PROGRAM PRG_Main
VAR
	bTestInput: BOOL;
	bTestOutput: BOOL;
	fbMachine: FB_ExampleMachine;
	fbStation1: FB_ExampleStation;
	fbStation2: FB_ExampleStation;
	fbStation3: FB_ExampleStation;
	fbStation4: FB_ExampleStation;
	bStart: BOOL;
	bAbort: BOOL;
	bReset: BOOL;
	bStop: BOOL;
	bSuspend: BOOL;
	fbDevice1: FB_ExampleDevice;
	fbDevice2: FB_ExampleDevice;
	fbDevice3: FB_ExampleDevice;
	fbDevice4: FB_ExampleDevice;
	bPoweredOn: BOOL;
//	FB_AdsDeviceAPI_0: FB_AdsDeviceAPI;
	FB_AdsDeviceAPI_0 : FB_AdsCommandRouter;
//	FB_AdsDeviceAPI_1 : FB_AdsCommandRouter;
	MyLaser1: FB_KeyenceLaserMarkerMDX2000;
	(* Database handler FB. *)
//	in_fbDataHandler: REFERENCE TO FB_Data;
	bConnectToLaserMarker: BOOL;
	bRes_LaserConnected: BOOL;
	bTestADSServer: BOOL;
	strTarget: T_MaxString;
	strCommand: T_MaxString;
	arrParams: T_ApiMethodParameters;
	MyResults: T_MaxString;
	bInterfaceTest : BOOL;
	temp: BOOL;
	bDisconnectFromLaserMarker: BOOL;
	bRes_LaserDisconnected: BOOL;
	bPeakCurrentProgramInLaser: BOOL;
	bRes_PeakCurrentProgramInLaser: BOOL;
	bSendProgramToLaser: BOOL;
	bRes_SendProgramtoLaser: BOOL;
	filepath : STRING;
	LaserMemoryLocation : INT;
	bSaveCurrentLaserProgramtoPC : BOOL;
	bRes_SaveCurrentLaserProgramtoPC: BOOL;
	LaserProgramFolderPath: STRING;
	bGetCurrentProgram : BOOL;
	bRes_GetCurrentProgram : BOOL;
	CurrentProgramName : T_MaxString;
	bStartMarking: BOOL;
	bRes_StartMarking: BOOL;
	bStopMarking: BOOL;
	bRes_StopMarking: BOOL;
	bClearLaserErrors: BOOL;
	bRes_ClearLaserErrors: BOOL;
	bUpdateProgramBlockInTheLaser: BOOL;
	bRes_UpdateProgramBlockInTheLaser: BOOL;
	_blockNumber: INT;
	_blockData: STRING;
	_blockType : BlockTypes;
	bGetLaserStatus: BOOL;
	bRes_GetLaserStatus: BOOL;
	_string_laserstatus : STRING;
	bGetLaserErrorStatus: BOOL;
	bRes_GetLaserErrorStatus: BOOL;
	_bIsLaserError : BOOL;
	bGetLaserActivatedStatus: BOOL;
	bRes_GetLaserActivatedStatus: BOOL;
	_bIsLaserActivated : BOOL;
	bGetLaserMarkingStatus: BOOL;
	bRes_GetLaserMarkingStatus: BOOL;
	_bIsLaserMarking : BOOL;
	bRes_Reset: BOOL;
	bResetErrors: BOOL;
	bUpdateProgramBlockMarkEnabledInTheLaser: BOOL;
	bRes_UpdateProgramBlockMarkEnabledInTheLaser: BOOL;
	_bool_markenabled : BOOL;
	_blockType_enum : BlockTypes;
	UpdateSingleBlockMarkEnabledIntheLaser_Success: BOOL;
	_bUpdateSingleBlockDataSuccess : BOOL;
	_bUpdateSingleBlockMarkEnabled_Success : BOOL;
	bUpdateAllMarkingInfo: BOOL;
	LastBlockToMark : INT;
	_OneTimeArrayBuild : BOOL := TRUE;
	BlockInfoArray : ARRAY [0..255] OF OneBlockInfo;
	bRes_UpdateAllMarkingInfo: BOOL;
	intIndex: INT;
	intIndex2 : INT;
	inst_intStep: INT := 0;
	_tempString : STRING;
	bRes_UpdateAllMarkInfo : ARRAY [0..255] OF BOOL;
	bUpdateAllMarkingInfo_MethodCall: BOOL;
	bRes_UpdateAllMarkingInfo_MethodCall: BOOL;
	fbDataHandler: FB_DataTracker;
	fbDataHandler2: FB_DataTracker;
	fbDatabaseCommandRouter: FB_AdsCommandRouter;
	_inst_bDataTransferred: BOOL;
	// (* Name of the parameters database transfer ID. *)
	in_strParametersDatabaseName: T_MaxString := 'GetLimits';
	in_strParametersDBNameLaserLimits_L1 : T_MaxString := 'GetLaserMarkingParams_L1';
	in_strParametersDBNameLaserLimits_L2 : T_MaxString := 'GetLaserMarkingParams_L2';
	in_strParametersDBNameLaserLimits_R1 : T_MaxString := 'GetLaserMarkingParams_R1';
	in_strParametersDBNameLaserLimits_R2 : T_MaxString := 'GetLaserMarkingParams_R2';	
	_inst_bLaserLimitsDataTransferred_L1 : BOOL;
	_inst_bLaserLimitsDataTransferred_L2 : BOOL;
	_inst_bLaserLimitsDataTransferred_R1 : BOOL;
	_inst_bLaserLimitsDataTransferred_R2 : BOOL;
	bGetLimitsFromDB : BOOL;
	bGetLaserParamsFromDB_L1 : BOOL;
	bGetLaserParamsFromDB_L2 : BOOL;
	bGetLaserParamsFromDB_R1 : BOOL;
	bGetLaserParamsFromDB_R2 : BOOL;
	bPerformPriorOp_Smart: BOOL;
	in_strParametersDBName_SmartWater : T_MaxString := 'GetPriorOPA';
	_inst_bPriorOp_Smart: BOOL;
	
	bPerformPriorOp_FFT: BOOL;
	in_strParametersDBName_FFTLaser_L1 : T_MaxString := 'LaserMarkCheckL1';
	_inst_bPriorOp_FFT: BOOL;
	
	Temp_CR_LOOKUP_NestL1 : INT;
	iLengthDataMatrixNestL1 : INT;
	ParamsArrayNestA : STRING;
	
	//MES Data Tracking Testing
//	fbDataHandler3: FB_MESDataTracking;
	bPerformGetLotInfoFromLotBarcode: BOOL;
	_inst_bGetLotInfo_LotBarcode: BOOL;
	in_strParamDBName_GetLotInfo: T_MaxString := 'GetLotInfo1';
	
	bPerformGetOpInfoFromOpBarcode: BOOL;
	in_strParamDBName_GetOpInfo: T_MaxString := 'GetOperatorInfo1';
	_inst_bGetOpInfo_OpBarcode: BOOL;
	
	bPerformStartLot : BOOL;
	_inst_bStartLot : BOOL;
	in_strParamDBName_StartLot : T_MaxString := 'StartLot1';
	
	bPerformGetProdLotComponents : BOOL;
	_inst_bGetProdLotComponents : BOOL;
	in_strParamDBName_GetProdLotComps : T_MaxString := 'GetProdLotComponents1';
	
	bPerformComponentValidation1 : BOOL;
	_inst_bCompValidation1 : BOOL;
	in_strParamDBName_Comp1Validation1 : T_MaxString := 'ComponentValidation1';
	
	bPerformComponentValidation2 : BOOL;
	_inst_bCompValidation2 : BOOL;
	in_strParamDBName_Comp1Validation2 : T_MaxString := 'ComponentValidation2';
	
	bPerformComponentValidation3 : BOOL;
	_inst_bCompValidation3 : BOOL;
	in_strParamDBName_Comp1Validation3 : T_MaxString := 'ComponentValidation3';
	
	bPerformGetMachineSettings : BOOL;
	_inst_bGetMachineSettings : BOOL;
	in_strParamDBName_GetMachSetting : T_MaxString := 'GetMachineSettings1';
	
	bPerformAddScrapCompByReason : BOOL;
	_inst_bAddScrapCompByReason : BOOL;
	in_strParamDBName_AddScrapCompByReason : T_MaxString := 'AddScrapComponentByReason1';
	
	bPerformEndLotComp : BOOL;
	_inst_bEndLotComp : BOOL;
	in_strParamDBName_EndLotComp : T_MaxString := 'EndLotComponent1';
	
	bPerformGetMachineDefects : BOOL;
	_inst_bGetMachineDefects : BOOL;
	in_strParamDBName_GetMachDefects : T_MaxString := 'GetMachineDefects1';

	//Testing Cohap Related Vars

	//Initialize Only	
	MyCohapTest : FB_COHAP;
	bInitializeCohapSystem: BOOL;
	bRes_CohapConnected: BOOL;

	//Execute RunImpMethods Only	;
	bExecuteRunImpMethods: BOOL;
	bRes_RunImpMethods: BOOL;

	//Set Current Device Instance
	bSetCurrentDevice_Cohap : BOOL;
	bRes_SetCurrentDevice : BOOL;
	//Input Params
	strDeviceName : STRING;
	
	//RunCommand
	bRunCommandCohapSystem : BOOL;
	bRes_RunCommand : BOOL;
	//Input Params
	strMethodName : STRING;
	RunCom_InpuParams : T_CohapParameterList;
	RunCom_ExpOutParamList : ARRAY[0..2] OF ReturnParamKVP;
	//Output Params
	RunCom_OutputParams : T_CohapParameterList;
	
	//DummyTest Dictionary Prep for RunCommand Execution
	RC_DT_InpPar : T_CohapParameterList;
	RC_DT_ExpOutPL : ARRAY[0..2] OF ReturnParamKVP;
	
	CohapMethodStrings : TMethodNames_Cohap;
	CohapMethodControls : TMethod_Controls;
//	fbCohapHandler1: FB_COHAP;

///////////////////////////////

	// For readSerialNumber
	readSerialNumber_inpuparams : T_CohapParameterList;// := [(strKey: 'channel', strValue: '1'), (), ()];
	readSerialNumber_expoutparamlist : ARRAY[0..2] OF ReturnParamKVP;// := [(VarName: 'serialnumber', DataType: DT_UINT), (), ()];
	readSerialNumber_outputparams : T_CohapParameterList;// := [(), (), ()];
	
	// For ReadDeviceOutput
	ReadDeviceOutput_inpuparams : T_CohapParameterList;// := [(strKey: 'Channel', strValue: '10'), (), ()];
	ReadDeviceOutput_expoutparamlist : ARRAY[0..2] OF ReturnParamKVP;// := [(VarName: 'Pressure', DataType: DT_STRING), (VarName: 'Temp', DataType: DT_STRING), ()];
	ReadDeviceOutput_outputparams : T_CohapParameterList;// := [(), (), ()];
	
	// For PowerUp
	PowerUp_inpuparams : T_CohapParameterList;// := [(strKey: 'channel', strValue: '1'), (strKey: 'supplyVoltage', strValue: '5.0'), ()];
	PowerUp_expoutparamlist : ARRAY[0..2] OF ReturnParamKVP;// := [(VarName: 'Vsupply', DataType: DT_DOUBLE), (VarName: 'current', DataType: DT_DOUBLE), ()];
	PowerUp_outputparams : T_CohapParameterList;// := [(), (), ()];
	
	// For PowerDown
	PowerDown_inpuparams : T_CohapParameterList;// := [(strKey: 'channel', strValue: '10'), (), ()];
	PowerDown_expoutparamlist : ARRAY[0..2] OF ReturnParamKVP;// := [(), (), ()];
	PowerDown_outputparams : T_CohapParameterList;// := [(), (), ()];
	
	// For initialize
//	initialize_inpuparams : T_CohapParameterList;// := [(), (), ()];
//	initialize_expoutparamlist : ARRAY[0..2] OF ReturnParamKVP;// := [(), (), ()];
//	initialize_outputparams : T_CohapParameterList;// := [(), (), ()];
	
	// For TestDummy
	TestDummy_inpuparams : T_CohapParameterList;// := [(strKey: 'channel', strValue: '10'), (), ()];
	TestDummy_expoutparamlist : ARRAY[0..2] OF ReturnParamKVP;// := [(VarName: 'serialno', DataType: DT_STRING), (), ()];
	TestDummy_outputparams : T_CohapParameterList;// := [(), (), ()];
	
	// For TestDummy2
	TestDummy2_inpuparams : T_CohapParameterList;// := [(strKey: 'channel', strValue: '10'), (), ()];
	TestDummy2_expoutparamlist : ARRAY[0..2] OF ReturnParamKVP;// := [(VarName: 'serialno', DataType: DT_STRING), (), ()];
	TestDummy2_outputparams : T_CohapParameterList;// := [(), (), ()];	
	
	// For init
	init_inpuparams : T_CohapParameterList;// := [(strKey: 'VSupply', strValue: '5.0'), (), ()];
	init_expoutparamlist : ARRAY[0..2] OF ReturnParamKVP;// := [(VarName: 'returnMsg', DataType: DT_STRING), (), ()];
	init_outputparams : T_CohapParameterList;// := [(), (), ()];
	
	// For getSICAndChannelCardVersions
	getSICAndChannelCardVersions_inpuparams : T_CohapParameterList;// := [(strKey: 'channel', strValue: '1'), (), ()];
	getSICAndChannelCardVersions_expoutparamlist : ARRAY[0..2] OF ReturnParamKVP;// := [(VarName: 'SICVersion', DataType: DT_STRING), (VarName: 'COHAPChannelCardVersion', DataType: DT_STRING), ()];
	getSICAndChannelCardVersions_outputparams : T_CohapParameterList;// := [(), (), ()];
	
	// For getDLLVersions
	getDLLVersions_inpuparams : T_CohapParameterList;// := [(), (), ()];
	getDLLVersions_expoutparamlist : ARRAY[0..2] OF ReturnParamKVP;// := [(VarName: 'DUT12133DLLVersion', DataType: DT_STRING), (VarName: 'MUPeT12133DLLVersion', DataType: DT_STRING), (VarName: 'HALDLLVersion', DataType: DT_STRING)];
	getDLLVersions_outputparams : T_CohapParameterList;// := [(), (), ()];
	
	// For initDUT
	initDUT_inpuparams : T_CohapParameterList;// := [(strKey: 'channel', strValue: '1'), (strKey: 'supplyVoltage', strValue: '5.0'), ()];
	initDUT_expoutparamlist : ARRAY[0..2] OF ReturnParamKVP;// := [(VarName: 'SICVersion', DataType: DT_STRING), (VarName: 'COHAPChannelCardVersion', DataType: DT_STRING), ()];
	initDUT_outputparams : T_CohapParameterList;// := [(), (), ()];



	TestDummyoutputParamsTest: T_ApiParameterList;
	TestDummy2_intResponse: INT;
	TestDummy2_floatResponse: LREAL;
END_VAR
VAR // added by the converter: edge detectors and wires of the graphical bodies
    _w1, _w2, _w3, _w4, _w5, _w6, _w7, _w8, _w9, _w10, _w11, _w12, _w13, _w14, _w15, _w16, _w17, _w18, _w19, _w20, _w21, _w22 : BOOL;
END_VAR

bTestOutput := bTestInput;

A_Machine();
//A_CohapLibraryTesting();
A_InitCohapMethodParams();
A_CohapLDTesting();

//A_Station1();
//A_Station2();
//A_Station3();
//A_Station4();
//bInterfaceTest := MyLaser1.fbApi.P_bDeviceInterfaceBusy;



//IF bPerformGetLotInfoFromLotBarcode THEN
//	_inst_bGetLotInfo_LotBarcode := fbDataHandler3.M_TransferData(in_strParamDBName_GetLotInfo);
//	IF _inst_bGetLotInfo_LotBarcode THEN
//		bPerformGetLotInfoFromLotBarcode := FALSE;
//	ELSIF fbDataHandler3.P_bError THEN 
//		bPerformGetLotInfoFromLotBarcode := FALSE;
//		fbDataHandler3.M_ClearError();
//	END_IF
//END_IF

//IF bPerformGetOpInfoFromOpBarcode THEN
//	_inst_bGetOpInfo_OpBarcode := fbDataHandler3.M_TransferData(in_strParamDBName_GetOpInfo);
//	IF _inst_bGetOpInfo_OpBarcode THEN
//		bPerformGetOpInfoFromOpBarcode := FALSE;
//	ELSIF fbDataHandler3.P_bError THEN 
//		bPerformGetOpInfoFromOpBarcode := FALSE;
//		fbDataHandler3.M_ClearError();
//	END_IF
//END_IF

//IF bPerformStartLot THEN
//	_inst_bStartLot := fbDataHandler3.M_TransferData(in_strParamDBName_StartLot);
//	IF _inst_bStartLot THEN
//		bPerformStartLot := FALSE;
//	ELSIF fbDataHandler3.P_bError THEN 
//		bPerformStartLot := FALSE;
//		fbDataHandler3.M_ClearError();
//	END_IF
//END_IF

//IF bPerformGetProdLotComponents THEN
//	_inst_bGetProdLotComponents := fbDataHandler3.M_TransferData(in_strParamDBName_GetProdLotComps);
//	IF _inst_bGetProdLotComponents THEN
//		bPerformGetProdLotComponents := FALSE;
//	ELSIF fbDataHandler3.P_bError THEN 
//		bPerformGetProdLotComponents := FALSE;
//		fbDataHandler3.M_ClearError();
//	END_IF
//END_IF


//IF bPerformComponentValidation1 THEN
//	_inst_bCompValidation1 := fbDataHandler3.M_TransferData(in_strParamDBName_Comp1Validation1);
//	IF _inst_bCompValidation1 THEN
//		bPerformComponentValidation1 := FALSE;
//	ELSIF fbDataHandler3.P_bError THEN 
//		bPerformComponentValidation1 := FALSE;
//		fbDataHandler3.M_ClearError();
//	END_IF
//END_IF

//IF bPerformComponentValidation2 THEN
//	_inst_bCompValidation2 := fbDataHandler3.M_TransferData(in_strParamDBName_Comp1Validation2);
//	IF _inst_bCompValidation2 THEN
//		bPerformComponentValidation2 := FALSE;
//	ELSIF fbDataHandler3.P_bError THEN 
//		bPerformComponentValidation2 := FALSE;
//		fbDataHandler3.M_ClearError();
//	END_IF
//END_IF

//IF bPerformComponentValidation3 THEN
//	_inst_bCompValidation3 := fbDataHandler3.M_TransferData(in_strParamDBName_Comp1Validation3);
//	IF _inst_bCompValidation3 THEN
//		bPerformComponentValidation3 := FALSE;
//	ELSIF fbDataHandler3.P_bError THEN 
//		bPerformComponentValidation3 := FALSE;
//		fbDataHandler3.M_ClearError();
//	END_IF
//END_IF

//IF bPerformGetMachineSettings THEN
//	_inst_bGetMachineSettings := fbDataHandler3.M_TransferData(in_strParamDBName_GetMachSetting);
//	IF _inst_bGetMachineSettings THEN
//		bPerformGetMachineSettings := FALSE;
//	ELSIF fbDataHandler3.P_bError THEN 
//		bPerformGetMachineSettings := FALSE;
//		fbDataHandler3.M_ClearError();
//	END_IF
//END_IF

//IF bPerformAddScrapCompByReason THEN
//	_inst_bAddScrapCompByReason := fbDataHandler3.M_TransferData(in_strParamDBName_AddScrapCompByReason);
//	IF _inst_bAddScrapCompByReason THEN
//		bPerformAddScrapCompByReason := FALSE;
//	ELSIF fbDataHandler3.P_bError THEN 
//		bPerformAddScrapCompByReason := FALSE;
//		fbDataHandler3.M_ClearError();
//	END_IF
//END_IF

//IF bPerformEndLotComp THEN
//	_inst_bEndLotComp := fbDataHandler3.M_TransferData(in_strParamDBName_EndLotComp);
//	IF _inst_bEndLotComp THEN
//		bPerformEndLotComp := FALSE;
//	ELSIF fbDataHandler3.P_bError THEN 
//		bPerformEndLotComp := FALSE;
//		fbDataHandler3.M_ClearError();
//	END_IF
//END_IF

//IF bPerformGetMachineDefects THEN
//	_inst_bGetMachineDefects := fbDataHandler3.M_TransferData(in_strParamDBName_GetMachDefects);
//	IF _inst_bGetMachineDefects THEN
//		bPerformGetMachineDefects := FALSE;
//	ELSIF fbDataHandler3.P_bError THEN 
//		bPerformGetMachineDefects := FALSE;
//		fbDataHandler3.M_ClearError();
//	END_IF
//END_IF

ACTION A_CohapLDTesting:
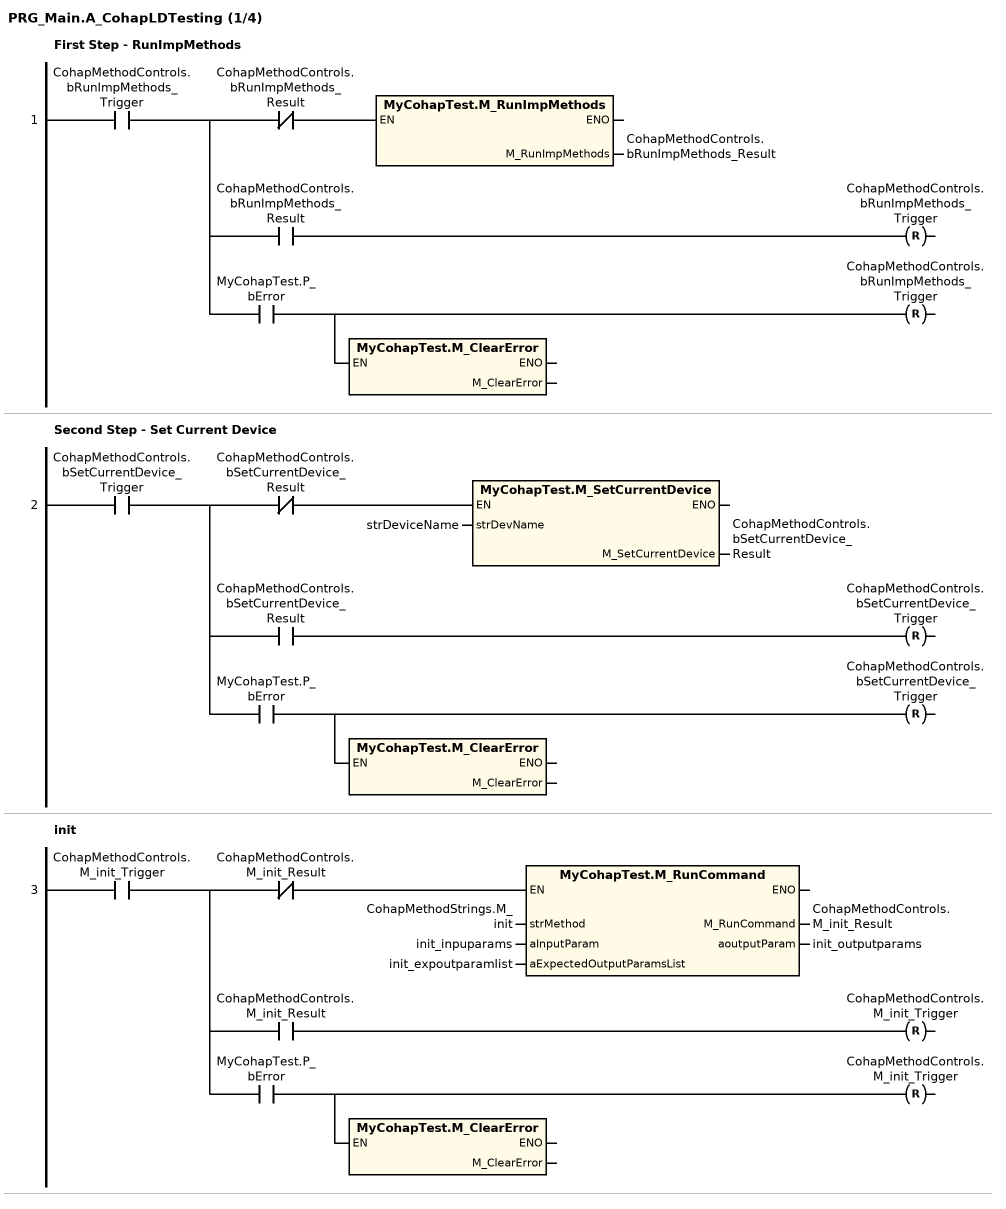
// NETWORK 1: First Step - RunImpMethods
_w1 := CohapMethodControls.bRunImpMethods_Trigger;
IF _w1 AND NOT CohapMethodControls.bRunImpMethods_Result THEN
    CohapMethodControls.bRunImpMethods_Result := MyCohapTest.M_RunImpMethods();
END_IF
CohapMethodControls.bRunImpMethods_Trigger R= _w1 AND CohapMethodControls.bRunImpMethods_Result;
_w2 := _w1 AND MyCohapTest.P_bError;
CohapMethodControls.bRunImpMethods_Trigger R= _w2;
IF _w2 THEN MyCohapTest.M_ClearError(); END_IF

// NETWORK 2: Second Step - Set Current Device
_w3 := CohapMethodControls.bSetCurrentDevice_Trigger;
IF _w3 AND NOT CohapMethodControls.bSetCurrentDevice_Result THEN
    CohapMethodControls.bSetCurrentDevice_Result := MyCohapTest.M_SetCurrentDevice(strDevName := strDeviceName);
END_IF
CohapMethodControls.bSetCurrentDevice_Trigger R= _w3 AND CohapMethodControls.bSetCurrentDevice_Result;
_w4 := _w3 AND MyCohapTest.P_bError;
CohapMethodControls.bSetCurrentDevice_Trigger R= _w4;
IF _w4 THEN MyCohapTest.M_ClearError(); END_IF

// NETWORK 3: init
_w5 := CohapMethodControls.M_init_Trigger;
IF _w5 AND NOT CohapMethodControls.M_init_Result THEN
    CohapMethodControls.M_init_Result := MyCohapTest.M_RunCommand(strMethod := CohapMethodStrings.M_init, aInputParam := init_inpuparams, aExpectedOutputParamsList := init_expoutparamlist, aoutputParam => init_outputparams);
END_IF
CohapMethodControls.M_init_Trigger R= _w5 AND CohapMethodControls.M_init_Result;
_w6 := _w5 AND MyCohapTest.P_bError;
CohapMethodControls.M_init_Trigger R= _w6;
IF _w6 THEN MyCohapTest.M_ClearError(); END_IF

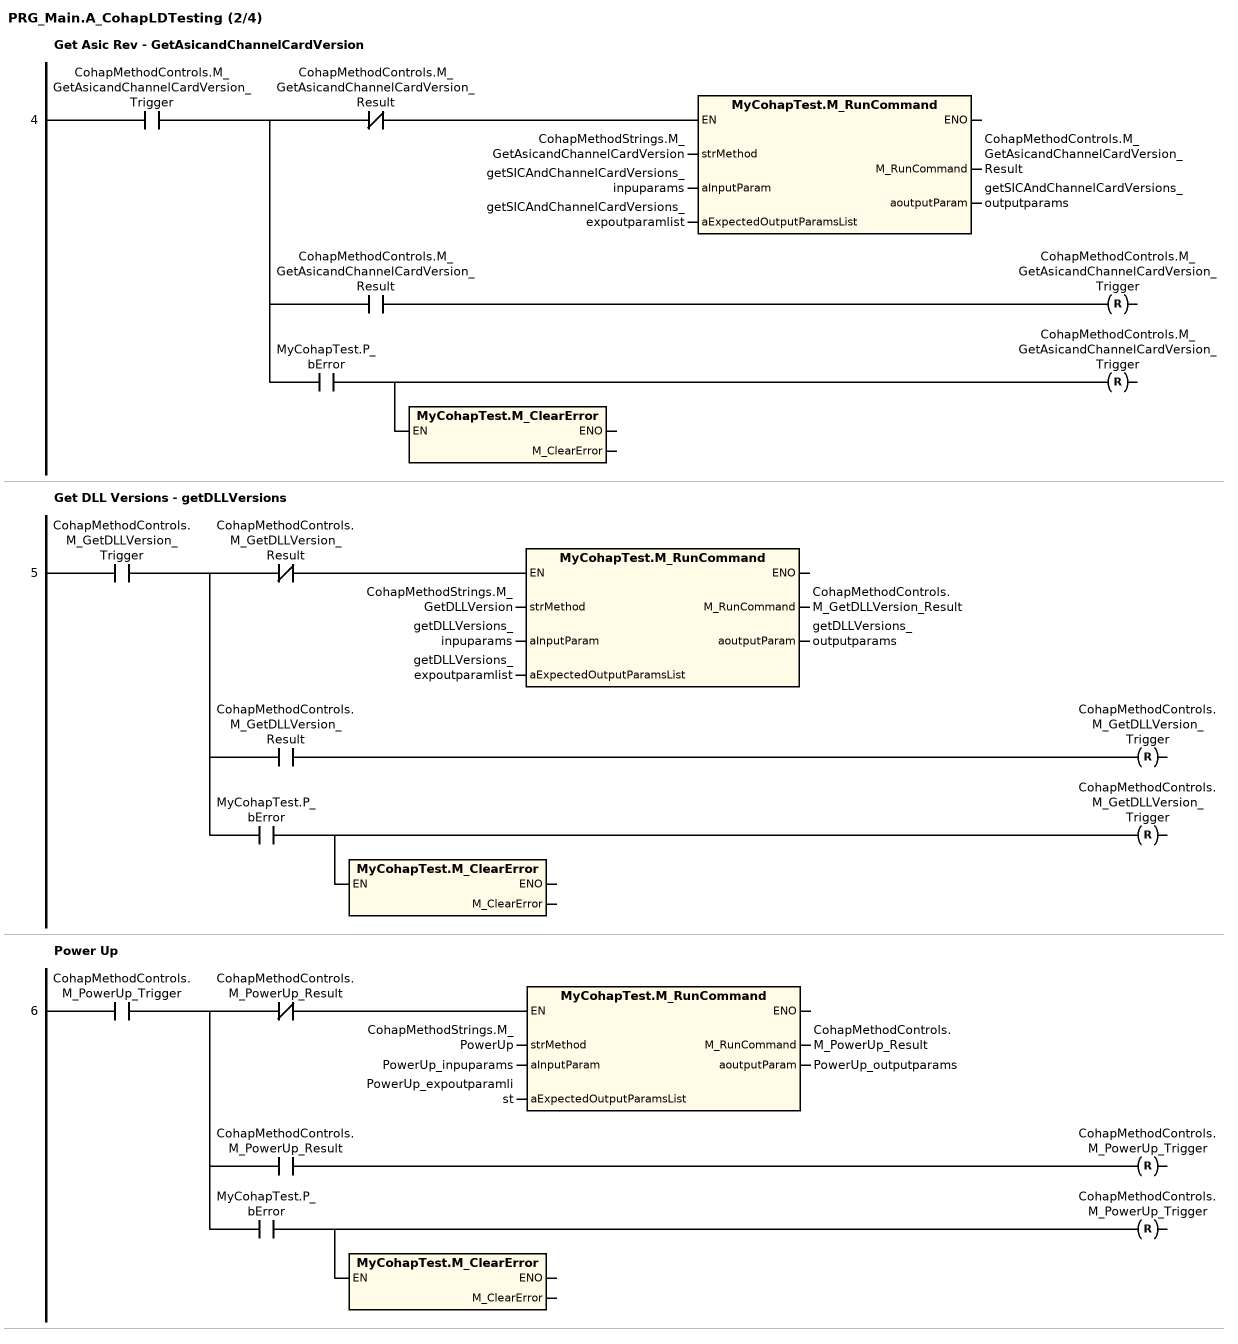
// NETWORK 4: Get Asic Rev - GetAsicandChannelCardVersion
_w7 := CohapMethodControls.M_GetAsicandChannelCardVersion_Trigger;
IF _w7 AND NOT CohapMethodControls.M_GetAsicandChannelCardVersion_Result THEN
    CohapMethodControls.M_GetAsicandChannelCardVersion_Result := MyCohapTest.M_RunCommand(strMethod := CohapMethodStrings.M_GetAsicandChannelCardVersion, aInputParam := getSICAndChannelCardVersions_inpuparams, aExpectedOutputParamsList := getSICAndChannelCardVersions_expoutparamlist, aoutputParam => getSICAndChannelCardVersions_outputparams);
END_IF
CohapMethodControls.M_GetAsicandChannelCardVersion_Trigger R= _w7 AND CohapMethodControls.M_GetAsicandChannelCardVersion_Result;
_w8 := _w7 AND MyCohapTest.P_bError;
CohapMethodControls.M_GetAsicandChannelCardVersion_Trigger R= _w8;
IF _w8 THEN MyCohapTest.M_ClearError(); END_IF

// NETWORK 5: Get DLL Versions - getDLLVersions
_w9 := CohapMethodControls.M_GetDLLVersion_Trigger;
IF _w9 AND NOT CohapMethodControls.M_GetDLLVersion_Result THEN
    CohapMethodControls.M_GetDLLVersion_Result := MyCohapTest.M_RunCommand(strMethod := CohapMethodStrings.M_GetDLLVersion, aInputParam := getDLLVersions_inpuparams, aExpectedOutputParamsList := getDLLVersions_expoutparamlist, aoutputParam => getDLLVersions_outputparams);
END_IF
CohapMethodControls.M_GetDLLVersion_Trigger R= _w9 AND CohapMethodControls.M_GetDLLVersion_Result;
_w10 := _w9 AND MyCohapTest.P_bError;
CohapMethodControls.M_GetDLLVersion_Trigger R= _w10;
IF _w10 THEN MyCohapTest.M_ClearError(); END_IF

// NETWORK 6: Power Up
_w11 := CohapMethodControls.M_PowerUp_Trigger;
IF _w11 AND NOT CohapMethodControls.M_PowerUp_Result THEN
    CohapMethodControls.M_PowerUp_Result := MyCohapTest.M_RunCommand(strMethod := CohapMethodStrings.M_PowerUp, aInputParam := PowerUp_inpuparams, aExpectedOutputParamsList := PowerUp_expoutparamlist, aoutputParam => PowerUp_outputparams);
END_IF
CohapMethodControls.M_PowerUp_Trigger R= _w11 AND CohapMethodControls.M_PowerUp_Result;
_w12 := _w11 AND MyCohapTest.P_bError;
CohapMethodControls.M_PowerUp_Trigger R= _w12;
IF _w12 THEN MyCohapTest.M_ClearError(); END_IF

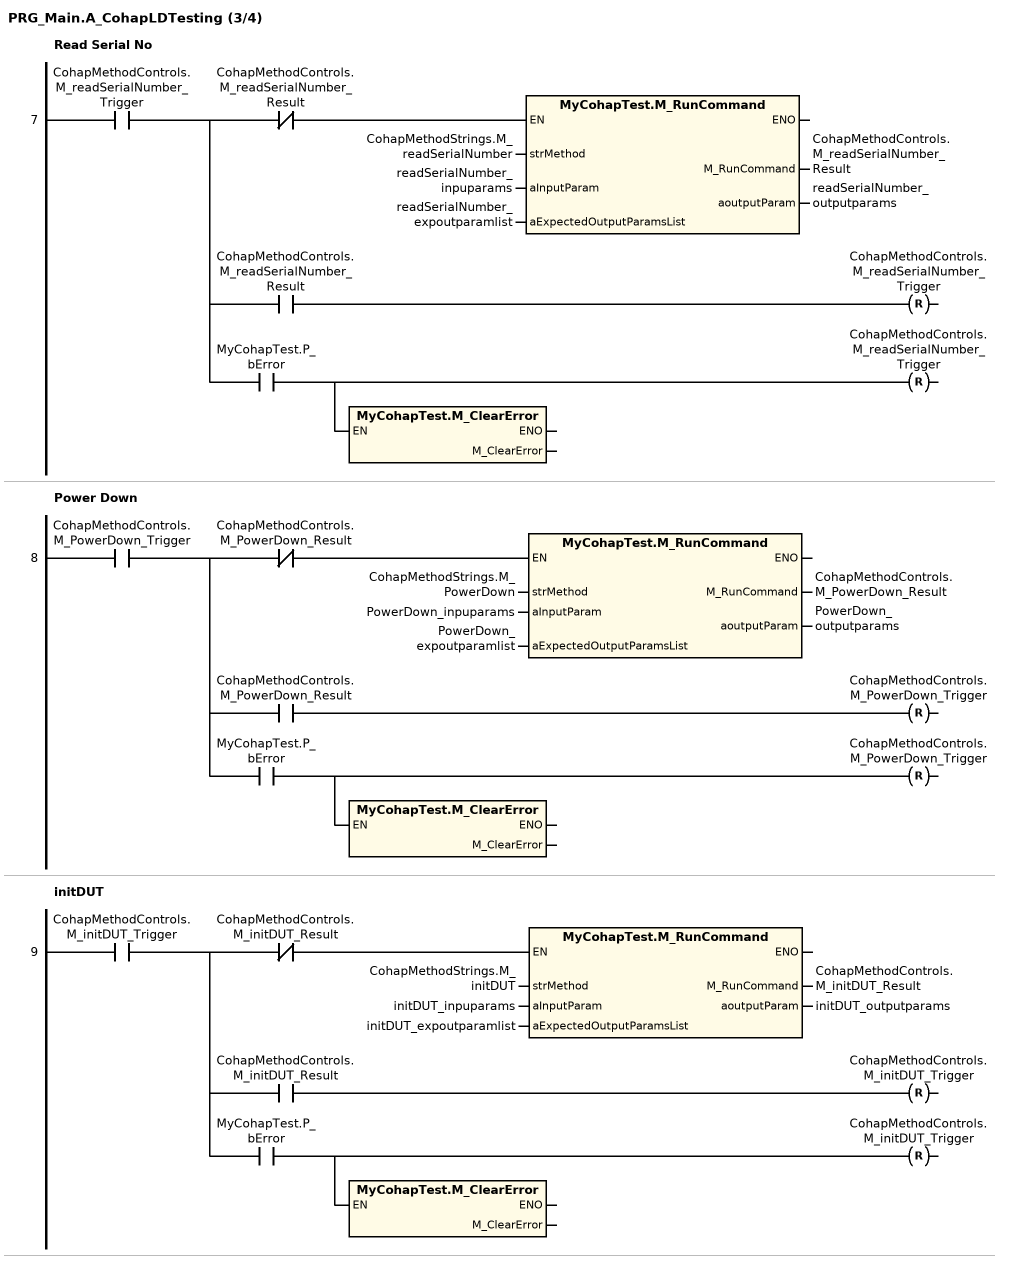
// NETWORK 7: Read Serial No
_w13 := CohapMethodControls.M_readSerialNumber_Trigger;
IF _w13 AND NOT CohapMethodControls.M_readSerialNumber_Result THEN
    CohapMethodControls.M_readSerialNumber_Result := MyCohapTest.M_RunCommand(strMethod := CohapMethodStrings.M_readSerialNumber, aInputParam := readSerialNumber_inpuparams, aExpectedOutputParamsList := readSerialNumber_expoutparamlist, aoutputParam => readSerialNumber_outputparams);
END_IF
CohapMethodControls.M_readSerialNumber_Trigger R= _w13 AND CohapMethodControls.M_readSerialNumber_Result;
_w14 := _w13 AND MyCohapTest.P_bError;
CohapMethodControls.M_readSerialNumber_Trigger R= _w14;
IF _w14 THEN MyCohapTest.M_ClearError(); END_IF

// NETWORK 8: Power Down
_w15 := CohapMethodControls.M_PowerDown_Trigger;
IF _w15 AND NOT CohapMethodControls.M_PowerDown_Result THEN
    CohapMethodControls.M_PowerDown_Result := MyCohapTest.M_RunCommand(strMethod := CohapMethodStrings.M_PowerDown, aInputParam := PowerDown_inpuparams, aExpectedOutputParamsList := PowerDown_expoutparamlist, aoutputParam => PowerDown_outputparams);
END_IF
CohapMethodControls.M_PowerDown_Trigger R= _w15 AND CohapMethodControls.M_PowerDown_Result;
_w16 := _w15 AND MyCohapTest.P_bError;
CohapMethodControls.M_PowerDown_Trigger R= _w16;
IF _w16 THEN MyCohapTest.M_ClearError(); END_IF

// NETWORK 9: initDUT
_w17 := CohapMethodControls.M_initDUT_Trigger;
IF _w17 AND NOT CohapMethodControls.M_initDUT_Result THEN
    CohapMethodControls.M_initDUT_Result := MyCohapTest.M_RunCommand(strMethod := CohapMethodStrings.M_initDUT, aInputParam := initDUT_inpuparams, aExpectedOutputParamsList := initDUT_expoutparamlist, aoutputParam => initDUT_outputparams);
END_IF
CohapMethodControls.M_initDUT_Trigger R= _w17 AND CohapMethodControls.M_initDUT_Result;
_w18 := _w17 AND MyCohapTest.P_bError;
CohapMethodControls.M_initDUT_Trigger R= _w18;
IF _w18 THEN MyCohapTest.M_ClearError(); END_IF

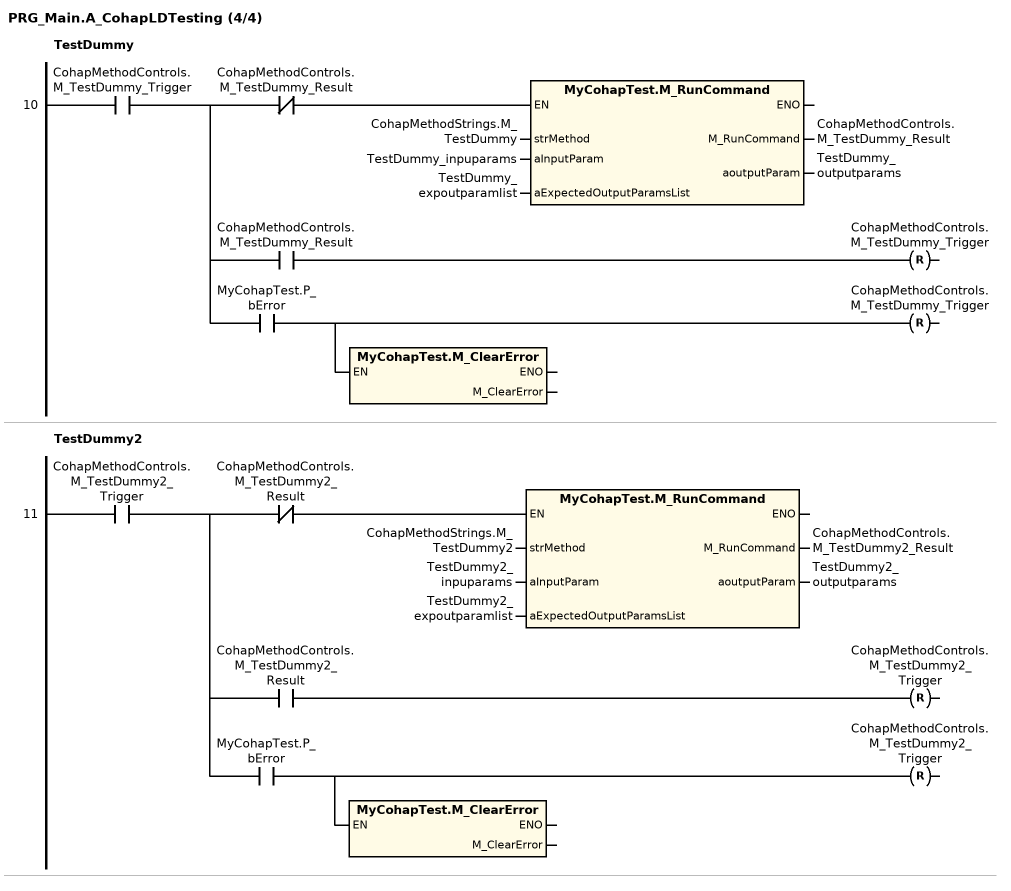
// NETWORK 10: TestDummy
_w19 := CohapMethodControls.M_TestDummy_Trigger;
IF _w19 AND NOT CohapMethodControls.M_TestDummy_Result THEN
    CohapMethodControls.M_TestDummy_Result := MyCohapTest.M_RunCommand(strMethod := CohapMethodStrings.M_TestDummy, aInputParam := TestDummy_inpuparams, aExpectedOutputParamsList := TestDummy_expoutparamlist, aoutputParam => TestDummy_outputparams);
END_IF
CohapMethodControls.M_TestDummy_Trigger R= _w19 AND CohapMethodControls.M_TestDummy_Result;
_w20 := _w19 AND MyCohapTest.P_bError;
CohapMethodControls.M_TestDummy_Trigger R= _w20;
IF _w20 THEN MyCohapTest.M_ClearError(); END_IF

// NETWORK 11: TestDummy2
_w21 := CohapMethodControls.M_TestDummy2_Trigger;
IF _w21 AND NOT CohapMethodControls.M_TestDummy2_Result THEN
    CohapMethodControls.M_TestDummy2_Result := MyCohapTest.M_RunCommand(strMethod := CohapMethodStrings.M_TestDummy2, aInputParam := TestDummy2_inpuparams, aExpectedOutputParamsList := TestDummy2_expoutparamlist, aoutputParam => TestDummy2_outputparams);
END_IF
CohapMethodControls.M_TestDummy2_Trigger R= _w21 AND CohapMethodControls.M_TestDummy2_Result;
_w22 := _w21 AND MyCohapTest.P_bError;
CohapMethodControls.M_TestDummy2_Trigger R= _w22;
IF _w22 THEN MyCohapTest.M_ClearError(); END_IF
END_ACTION

ACTION A_CohapLibraryTesting:
//IF bInitializeCohapSystem THEN
//	bRes_CohapConnected := MyCohapTest.M_init(1);
//	IF bRes_CohapConnected THEN
//	//Add some timer based logic to do error handling.
//		bInitializeCohapSystem := FALSE;
//	ELSIF MyCohapTest.P_bError THEN
//		bInitializeCohapSystem := FALSE;
//		MyCohapTest.M_ClearError();
//	END_IF
//END_IF

//IF bExecuteRunImpMethods THEN
//	bRes_RunImpMethods := MyCohapTest.M_RunImpMethods();
//	IF bRes_RunImpMethods THEN
//	//Add some timer based logic to do error handling.
//		bExecuteRunImpMethods := FALSE;
//	ELSIF MyCohapTest.P_bError THEN
//		bExecuteRunImpMethods := FALSE;
//		MyCohapTest.M_ClearError();
//	END_IF
//END_IF


//IF bSetCurrentDevice_Cohap THEN
//	bRes_SetCurrentDevice := MyCohapTest.M_SetCurrentDevice(strDeviceName);
//	IF bRes_SetCurrentDevice THEN
//	//Add some timer based logic to do error handling.
//		bSetCurrentDevice_Cohap := FALSE;
//	ELSIF MyCohapTest.P_bError THEN
//		bSetCurrentDevice_Cohap := FALSE;
//		MyCohapTest.M_ClearError();
//	END_IF
//END_IF


//RC_DT_InpPar[1].strKey := 'channel';
//RC_DT_InpPar[1].strValue := '123';

////RC_DT_InpPar[1].strKey := '';
////RC_DT_InpPar[1].strValue := '';

//RC_DT_ExpOutPL[1].VarName := 'serialno';
//RC_DT_ExpOutPL[1].DataType := E_DataType.DT_STRING;

////RC_DT_ExpOutPL[1].VarName := '';
////RC_DT_ExpOutPL[1].DataType := E_DataType.DT_BOOL;


//IF bRunCommandCohapSystem THEN
//	bRes_RunCommand := MyCohapTest.M_RunCommand(strMethodName, RunCom_InpuParams, RunCom_ExpOutParamList, aoutputParam => RunCom_OutputParams );
//	IF bRes_RunCommand THEN
//	//Add some timer based logic to do error handling.
//		bRunCommandCohapSystem := FALSE;
//	ELSIF MyCohapTest.P_bError THEN
//		bRunCommandCohapSystem := FALSE;
//		MyCohapTest.M_ClearError();
//	END_IF
//END_IF
END_ACTION

ACTION A_InitCohapMethodParams:
strDeviceName := 'Device12133';

readSerialNumber_inpuparams[0].strKey := 'channel';
readSerialNumber_inpuparams[0].strValue := '1';
readSerialNumber_inpuparams[1].strKey := '';
readSerialNumber_inpuparams[1].strValue := '';
readSerialNumber_inpuparams[2].strKey := '';
readSerialNumber_inpuparams[2].strValue := '';

readSerialNumber_expoutparamlist[0].DataType := E_DataType.DT_UINT;
readSerialNumber_expoutparamlist[0].VarName := 'serialnumber';
readSerialNumber_expoutparamlist[1].DataType := E_DataType.DT_STRING;
readSerialNumber_expoutparamlist[1].VarName := '';
readSerialNumber_expoutparamlist[2].DataType := E_DataType.DT_STRING;
readSerialNumber_expoutparamlist[2].VarName := '';


ReadDeviceOutput_inpuparams[0].strKey := 'channel';
ReadDeviceOutput_inpuparams[0].strValue := '1';
ReadDeviceOutput_inpuparams[1].strKey := '';
ReadDeviceOutput_inpuparams[1].strValue := '';
ReadDeviceOutput_inpuparams[2].strKey := '';
ReadDeviceOutput_inpuparams[2].strValue := '';

ReadDeviceOutput_expoutparamlist[0].DataType := E_DataType.DT_STRING;
ReadDeviceOutput_expoutparamlist[0].VarName := '';
ReadDeviceOutput_expoutparamlist[1].DataType := E_DataType.DT_STRING;
ReadDeviceOutput_expoutparamlist[1].VarName := '';
ReadDeviceOutput_expoutparamlist[2].DataType := E_DataType.DT_STRING;
ReadDeviceOutput_expoutparamlist[2].VarName := '';


PowerUp_inpuparams[0].strKey := 'channel';
PowerUp_inpuparams[0].strValue := '1';
PowerUp_inpuparams[1].strKey := 'supplyVoltage';
PowerUp_inpuparams[1].strValue := '5.0';
PowerUp_inpuparams[2].strKey := '';
PowerUp_inpuparams[2].strValue := '';

PowerUp_expoutparamlist[0].DataType := E_DataType.DT_DOUBLE;
PowerUp_expoutparamlist[0].VarName := 'Vsupply';
PowerUp_expoutparamlist[1].DataType := E_DataType.DT_DOUBLE;
PowerUp_expoutparamlist[1].VarName := 'current';
PowerUp_expoutparamlist[2].DataType := E_DataType.DT_STRING;
PowerUp_expoutparamlist[2].VarName := '';

PowerDown_inpuparams[0].strKey := 'channel';
PowerDown_inpuparams[0].strValue := '1';
PowerDown_inpuparams[1].strKey := '';
PowerDown_inpuparams[1].strValue := '';
PowerDown_inpuparams[2].strKey := '';
PowerDown_inpuparams[2].strValue := '';

PowerDown_expoutparamlist[0].DataType := E_DataType.DT_STRING;
PowerDown_expoutparamlist[0].VarName := '';
PowerDown_expoutparamlist[1].DataType := E_DataType.DT_STRING;
PowerDown_expoutparamlist[1].VarName := '';
PowerDown_expoutparamlist[2].DataType := E_DataType.DT_STRING;
PowerDown_expoutparamlist[2].VarName := '';

TestDummy_inpuparams[0].strKey := 'channel';
TestDummy_inpuparams[0].strValue := '1';
TestDummy_inpuparams[1].strKey := 'bInput';
TestDummy_inpuparams[1].strValue := 'FALSE';
TestDummy_inpuparams[2].strKey := '';
TestDummy_inpuparams[2].strValue := '';

TestDummy_expoutparamlist[0].DataType := E_DataType.DT_STRING;
TestDummy_expoutparamlist[0].VarName := 'serialno';
TestDummy_expoutparamlist[1].DataType := E_DataType.DT_DOUBLE;
TestDummy_expoutparamlist[1].VarName := 'Voltage';
TestDummy_expoutparamlist[2].DataType := E_DataType.DT_BOOL;
TestDummy_expoutparamlist[2].VarName := 'MethodResponse';

TestDummy2_inpuparams[0].strKey := 'channel';
TestDummy2_inpuparams[0].strValue := '1';
TestDummy2_inpuparams[1].strKey := 'Input2';
TestDummy2_inpuparams[1].strValue := 'dummyimput2';
TestDummy2_inpuparams[2].strKey := '';
TestDummy2_inpuparams[2].strValue := '';

TestDummy2_expoutparamlist[0].DataType := E_DataType.DT_INT;
TestDummy2_expoutparamlist[0].VarName := 'output1';
TestDummy2_expoutparamlist[1].DataType := E_DataType.DT_STRING;
TestDummy2_expoutparamlist[1].VarName := 'output2';
TestDummy2_expoutparamlist[2].DataType := E_DataType.DT_STRING;
TestDummy2_expoutparamlist[2].VarName := '';

init_inpuparams[0].strKey := 'VSupply';
init_inpuparams[0].strValue := '5.0';
init_inpuparams[1].strKey := '';
init_inpuparams[1].strValue := '';
init_inpuparams[2].strKey := '';
init_inpuparams[2].strValue := '';

init_expoutparamlist[0].DataType := E_DataType.DT_STRING;
init_expoutparamlist[0].VarName := 'returnMsg';
init_expoutparamlist[1].DataType := E_DataType.DT_STRING;
init_expoutparamlist[1].VarName := '';
init_expoutparamlist[2].DataType := E_DataType.DT_STRING;
init_expoutparamlist[2].VarName := '';

getSICAndChannelCardVersions_inpuparams[0].strKey := 'channel';
getSICAndChannelCardVersions_inpuparams[0].strValue := '1';
getSICAndChannelCardVersions_inpuparams[1].strKey := '';
getSICAndChannelCardVersions_inpuparams[1].strValue := '';
getSICAndChannelCardVersions_inpuparams[2].strKey := '';
getSICAndChannelCardVersions_inpuparams[2].strValue := '';

getSICAndChannelCardVersions_expoutparamlist[0].DataType := E_DataType.DT_STRING;
getSICAndChannelCardVersions_expoutparamlist[0].VarName := 'SICVersion';
getSICAndChannelCardVersions_expoutparamlist[1].DataType := E_DataType.DT_STRING;
getSICAndChannelCardVersions_expoutparamlist[1].VarName := 'COHAPChannelCardVersion';
getSICAndChannelCardVersions_expoutparamlist[2].DataType := E_DataType.DT_STRING;
getSICAndChannelCardVersions_expoutparamlist[2].VarName := '';

getDLLVersions_inpuparams[0].strKey := '';
getDLLVersions_inpuparams[0].strValue := '';
getDLLVersions_inpuparams[1].strKey := '';
getDLLVersions_inpuparams[1].strValue := '';
getDLLVersions_inpuparams[2].strKey := '';
getDLLVersions_inpuparams[2].strValue := '';

getDLLVersions_expoutparamlist[0].DataType := E_DataType.DT_STRING;
getDLLVersions_expoutparamlist[0].VarName := 'DUT12133DLLVersion';
getDLLVersions_expoutparamlist[1].DataType := E_DataType.DT_STRING;
getDLLVersions_expoutparamlist[1].VarName := 'MUPeT12133DLLVersion';
getDLLVersions_expoutparamlist[2].DataType := E_DataType.DT_STRING;
getDLLVersions_expoutparamlist[2].VarName := 'HALDLLVersion';


initDUT_inpuparams[0].strKey := 'channel';
initDUT_inpuparams[0].strValue := '1';
initDUT_inpuparams[1].strKey := 'supplyVoltage';
initDUT_inpuparams[1].strValue := '5.0';
initDUT_inpuparams[2].strKey := '';
initDUT_inpuparams[2].strValue := '';

initDUT_expoutparamlist[0].DataType := E_DataType.DT_STRING;
initDUT_expoutparamlist[0].VarName := '';
initDUT_expoutparamlist[1].DataType := E_DataType.DT_STRING;
initDUT_expoutparamlist[1].VarName := '';
initDUT_expoutparamlist[2].DataType := E_DataType.DT_STRING;
initDUT_expoutparamlist[2].VarName := '';
END_ACTION

ACTION A_LaserMarkingParams:
//IF bConnectToLaserMarker THEN
//	bRes_LaserConnected := MyLaser1.M_Connect();
//	IF bRes_LaserConnected THEN
//	//Add some timer based logic to do error handling.
//		bConnectToLaserMarker := FALSE;
//	ELSIF MyLaser1.P_bError THEN
//		bConnectToLaserMarker := FALSE;
//		MyLaser1.M_ClearError();
//	END_IF
//END_IF


//IF bDisconnectFromLaserMarker THEN
//	bRes_LaserDisconnected := MyLaser1.M_Disconnect();
//	IF bRes_LaserDisconnected THEN
//		bDisconnectFromLaserMarker := FALSE;
//	ELSIF MyLaser1.P_bError THEN
//		bDisconnectFromLaserMarker := FALSE;
//		MyLaser1.M_ClearError();
//	END_IF
//END_IF


//IF bPeakCurrentProgramInLaser THEN
//	bRes_PeakCurrentProgramInLaser := MyLaser1.M_PeakCurrentProgram();
//	IF bRes_PeakCurrentProgramInLaser THEN
//		bPeakCurrentProgramInLaser := FALSE;
//	ELSIF MyLaser1.P_bError THEN
//		bPeakCurrentProgramInLaser := FALSE;
//		MyLaser1.M_ClearError();
//	END_IF
//END_IF


//IF bSendProgramToLaser THEN
//	bRes_SendProgramtoLaser := MyLaser1.M_SendProgramtoLaser(filepath,LaserMemoryLocation);
//	IF bRes_SendProgramtoLaser THEN
//		bSendProgramToLaser := FALSE;
//	ELSIF MyLaser1.P_bError THEN
//		bSendProgramToLaser := FALSE;
//		MyLaser1.M_ClearError();
//	END_IF
//END_IF

//IF bSaveCurrentLaserProgramtoPC THEN
//	bRes_SaveCurrentLaserProgramtoPC := MyLaser1.M_SaveCurrentLaserProgramtoPC(LaserProgramFolderPath, out_bool_SaveProgramToPC_Success => SaveCurrentLaserProgramToPCSuccess);
//	IF bRes_SaveCurrentLaserProgramtoPC THEN
////		SaveCurrentLaserProgramToPCSuccess := MyLaser1
//		bSaveCurrentLaserProgramtoPC := FALSE;
//	ELSIF MyLaser1.P_bError THEN
//		bSaveCurrentLaserProgramtoPC := FALSE;
//		MyLaser1.M_ClearError();
//	END_IF
//END_IF

//IF bGetCurrentProgram THEN
//	bRes_GetCurrentProgram := MyLaser1.M_GetCurrentProgram(strCurrentProgram => CurrentProgramName);
//	IF bRes_GetCurrentProgram THEN
//		bGetCurrentProgram := FALSE;
//	ELSIF MyLaser1.P_bError THEN
//		bGetCurrentProgram := FALSE;
//		MyLaser1.M_ClearError();
//	END_IF
//END_IF

//IF bStartMarking THEN
//	bRes_StartMarking := MyLaser1.M_StartMarking();
//	IF bRes_StartMarking THEN
//		bStartMarking := FALSE;
//	ELSIF MyLaser1.P_bError THEN
//		bStartMarking := FALSE;
//		MyLaser1.M_ClearError();
//	END_IF
//END_IF

//IF bStopMarking THEN
//	bRes_StopMarking := MyLaser1.M_StopMarking();
//	IF bRes_StopMarking THEN
//		bStopMarking := FALSE;
//	ELSIF MyLaser1.P_bError THEN
//		bStopMarking := FALSE;
//		MyLaser1.M_ClearError();
//	END_IF
//END_IF

//IF bResetErrors THEN
//	bRes_Reset := MyLaser1.M_Reset();
//	IF bRes_Reset THEN
//		bResetErrors := FALSE;
//	ELSIF MyLaser1.P_bError THEN
//		bResetErrors := FALSE;
//		MyLaser1.M_ClearError();
//	END_IF
//END_IF

////IF bUpdateProgramBlockInTheLaser THEN
////	bRes_UpdateProgramBlockInTheLaser := MyLaser1.M_UpdateSingleProgramBlockData(LaserMemoryLocation, _blockNumber, _blockData, _blockType, out_bool_UpdateData_Success => _bUpdateSingleBlockDataSuccess);
////	IF bRes_UpdateProgramBlockInTheLaser THEN
////		bUpdateProgramBlockInTheLaser := FALSE;
////	ELSIF MyLaser1.P_bError THEN
////		bUpdateProgramBlockInTheLaser := FALSE;
////		MyLaser1.M_ClearError();
////	END_IF
////END_IF

//IF bUpdateProgramBlockInTheLaser THEN
//	bRes_UpdateProgramBlockInTheLaser := MyLaser1.M_UpdateSingleBlockMarkingInformation(_blockNumber, _blockData, _bool_markenabled);
//	IF bRes_UpdateProgramBlockInTheLaser THEN
//		bUpdateProgramBlockInTheLaser := FALSE;
//	ELSIF MyLaser1.P_bError THEN
//		bUpdateProgramBlockInTheLaser := FALSE;
//		MyLaser1.M_ClearError();
//	END_IF
//END_IF

//IF bUpdateProgramBlockMarkEnabledInTheLaser THEN
//	bRes_UpdateProgramBlockMarkEnabledInTheLaser := MyLaser1.M_UpdateSingleProgramBlockMarkEnabled( LaserProgramMemoryLocation := LaserMemoryLocation, BlockNumber := _blockNumber, BlockType := _blockType ,MarkEnabled := _bool_markenabled ,out_bool_MarkEnabled_Success => _bUpdateSingleBlockMarkEnabled_Success);
//	IF bRes_UpdateProgramBlockMarkEnabledInTheLaser THEN
//		bUpdateProgramBlockMarkEnabledInTheLaser := FALSE;
//	ELSIF MyLaser1.P_bError THEN
//		bUpdateProgramBlockMarkEnabledInTheLaser := FALSE;
//		MyLaser1.M_ClearError();
//	END_IF
//END_IF

//IF bGetLaserStatus THEN
//	bRes_GetLaserStatus := MyLaser1.M_GetLaserStatus( out_string_laserStatus => _string_laserstatus);
//	IF bRes_GetLaserStatus THEN
//		bGetLaserStatus := FALSE;
//	ELSIF MyLaser1.P_bError THEN
//		bGetLaserStatus := FALSE;
//		MyLaser1.M_ClearError();
//	END_IF
//END_IF

//IF bGetLaserErrorStatus THEN
//	bRes_GetLaserErrorStatus := MyLaser1.M_GetLaserErrorStatus( out_bool_IsLaserError => _bIsLaserError);
//	IF bRes_GetLaserErrorStatus THEN
//		bGetLaserErrorStatus := FALSE;
//	ELSIF MyLaser1.P_bError THEN
//		bGetLaserErrorStatus := FALSE;
//		MyLaser1.M_ClearError();
//	END_IF
//END_IF

//IF bGetLaserActivatedStatus THEN
//	bRes_GetLaserActivatedStatus := MyLaser1.M_GetLaserActivatedStatus( out_IsLaserActivated => _bIsLaserActivated);
//	IF bRes_GetLaserActivatedStatus THEN
//		bGetLaserActivatedStatus := FALSE;
//	ELSIF MyLaser1.P_bError THEN
//		bGetLaserActivatedStatus := FALSE;
//		MyLaser1.M_ClearError();
//	END_IF
//END_IF

//IF bGetLaserMarkingStatus THEN
//	bRes_GetLaserMarkingStatus := MyLaser1.M_GetLaserMarkingStatus( out_bool_IsLaserMarking => _bIsLaserMarking);
//	IF bRes_GetLaserMarkingStatus THEN
//		bGetLaserMarkingStatus := FALSE;
//	ELSIF MyLaser1.P_bError THEN
//		bGetLaserMarkingStatus := FALSE;
//		MyLaser1.M_ClearError();
//	END_IF
//END_IF

//IF _OneTimeArrayBuild THEN
//	FOR intIndex2 := 0 TO 255 DO
//		IF intIndex2 <= LastBlockToMark THEN
//			BlockInfoArray[intIndex2].MarkEnabled := TRUE;
//			_tempString := CONCAT('Block', INT_TO_STRING(intIndex2));
//			BlockInfoArray[intIndex2].BlockText := _tempString;
//		ELSE
//			BlockInfoArray[intIndex2].MarkEnabled := FALSE;	
//			BlockInfoArray[intIndex2].BlockText := '';
//		END_IF
//	END_FOR
//	_OneTimeArrayBuild := FALSE;
//END_IF

//IF bUpdateAllMarkingInfo_MethodCall THEN
//	bRes_UpdateAllMarkingInfo_MethodCall := MyLaser1.M_UpdateAllMarkingInformation(LastBlockToMark);
//	bUpdateAllMarkingInfo_MethodCall := FALSE;
//END_IF
//IF MyLaser1.P_bError THEN
//	bUpdateAllMarkingInfo_MethodCall := FALSE;
//	MyLaser1.M_ClearError();
//END_IF

//IF bUpdateAllMarkingInfo THEN
//	CASE inst_intStep OF
//		0: //Check for errors and Integer value which we are gonna run the update single block information
//				IF MyLaser1.P_bError THEN
//					inst_intStep := 0;
//					bUpdateAllMarkingInfo := FALSE;
//				ELSE
//					inst_intStep := 10;
//				END_IF
//		10: // Run the M_UpdateSingleBlockMarkingInformation Command
//				bRes_UpdateAllMarkInfo[intIndex] := MyLaser1.M_UpdateSingleBlockMarkingInformation(intIndex ,BlockInfoArray[intIndex].BlockText, BlockInfoArray[intIndex].MarkEnabled);
//				IF bRes_UpdateAllMarkInfo[intIndex] THEN 
//					inst_intStep := 20;
//				ELSIF MyLaser1.P_bError THEN
//					inst_intStep := 0;
//					intIndex :=0;
//					bUpdateAllMarkingInfo := FALSE;
//				END_IF
//		20: // Check if the M_UpdateSingleBlockMarkingInformation command failed or passed
//				IF bRes_UpdateAllMarkInfo[LastBlockToMark] OR NOT bRes_UpdateAllMarkInfo[intIndex] OR (intIndex = LastBlockToMark) THEN //This means we reached the final element update
//					bUpdateAllMarkingInfo := FALSE;
//					intIndex :=0;
//					inst_intStep := 0;
//				ELSIF bRes_UpdateAllMarkInfo[intIndex] THEN
//					inst_intStep := 0;
//					intIndex := intIndex + 1;
//				ELSIF MyLaser1.P_bError THEN
//					bUpdateAllMarkingInfo := FALSE;
//					MyLaser1.M_ClearError();	
//				END_IF			
//	END_CASE
//END_IF

//IF bGetLimitsFromDB THEN
//	_inst_bDataTransferred := fbDataHandler.M_TransferData(in_strParametersDatabaseName);
//	IF _inst_bDataTransferred THEN
//		bGetLimitsFromDB := FALSE;
//	ELSIF fbDataHandler.P_bError THEN
//		bGetLimitsFromDB := FALSE;
//		fbDataHandler.M_ClearError();
//	END_IF
//END_IF

//IF bGetLaserParamsFromDB_L1 THEN
//	_inst_bLaserLimitsDataTransferred_L1 := fbDataHandler.M_TransferData(in_strParametersDBNameLaserLimits_L1);
//	IF _inst_bLaserLimitsDataTransferred_L1 THEN
//		bGetLaserParamsFromDB_L1 := FALSE;
//		ELSIF fbDataHandler.P_bError THEN
//			bGetLaserParamsFromDB_L1 := FALSE;
//			fbDataHandler.M_ClearError();
//	END_IF
//END_IF

//IF bGetLaserParamsFromDB_L2 THEN
//	_inst_bLaserLimitsDataTransferred_L2 := fbDataHandler.M_TransferData(in_strParametersDBNameLaserLimits_L2);
//	IF _inst_bLaserLimitsDataTransferred_L2 THEN
//		bGetLaserParamsFromDB_L2 := FALSE;
//		ELSIF fbDataHandler.P_bError THEN
//			bGetLaserParamsFromDB_L2 := FALSE;
//			fbDataHandler.M_ClearError();
//	END_IF
//END_IF

//IF bGetLaserParamsFromDB_R1 THEN
//	_inst_bLaserLimitsDataTransferred_R1 := fbDataHandler.M_TransferData(in_strParametersDBNameLaserLimits_R1);
//	IF _inst_bLaserLimitsDataTransferred_R1 THEN
//		bGetLaserParamsFromDB_R1 := FALSE;
//		ELSIF fbDataHandler.P_bError THEN
//			bGetLaserParamsFromDB_R1 := FALSE;
//			fbDataHandler.M_ClearError();
//	END_IF
//END_IF

//IF bGetLaserParamsFromDB_R2 THEN
//	_inst_bLaserLimitsDataTransferred_R2 := fbDataHandler.M_TransferData(in_strParametersDBNameLaserLimits_R2);
//	IF _inst_bLaserLimitsDataTransferred_R2 THEN
//		bGetLaserParamsFromDB_R2 := FALSE;
//		ELSIF fbDataHandler.P_bError THEN
//			bGetLaserParamsFromDB_R2 := FALSE;
//			fbDataHandler.M_ClearError();
//	END_IF
//END_IF

//IF bPerformPriorOp_Smart THEN
//	_inst_bPriorOp_Smart := fbDataHandler2.M_TransferData(in_strParametersDBName_SmartWater);
//	IF _inst_bPriorOp_Smart THEN
//		bPerformPriorOp_Smart := FALSE;
//	ELSIF fbDataHandler2.P_bError THEN 
//		bPerformPriorOp_Smart := FALSE;
//		fbDataHandler2.M_ClearError();
//	END_IF
//END_IF

//IF bPerformPriorOp_FFT THEN
//	_inst_bPriorOp_FFT := fbDataHandler.M_TransferData(in_strParametersDBName_FFTLaser_L1);
//	IF _inst_bPriorOp_FFT THEN
//		bPerformPriorOp_FFT := FALSE;
//	ELSIF fbDataHandler.P_bError THEN 
//		bPerformPriorOp_FFT := FALSE;
//		fbDataHandler.M_ClearError();
//	END_IF
//END_IF

//Temp_CR_LOOKUP_NestL1 := FIND('GV354-006:220705-141019_CR','_CR');
//iLengthDataMatrixNestL1 := LEN('GV354-006:220705-141019_CR');
//IF  (Temp_CR_LOOKUP_NestL1 > 0) THEN
//	ParamsArrayNestA := REPLACE('GV354-006:220705-141019_CR', concat(' CR ' , '0.023456'),6,iLengthDataMatrixNestL1 - 2);
//END_IF
END_ACTION

ACTION A_Machine:
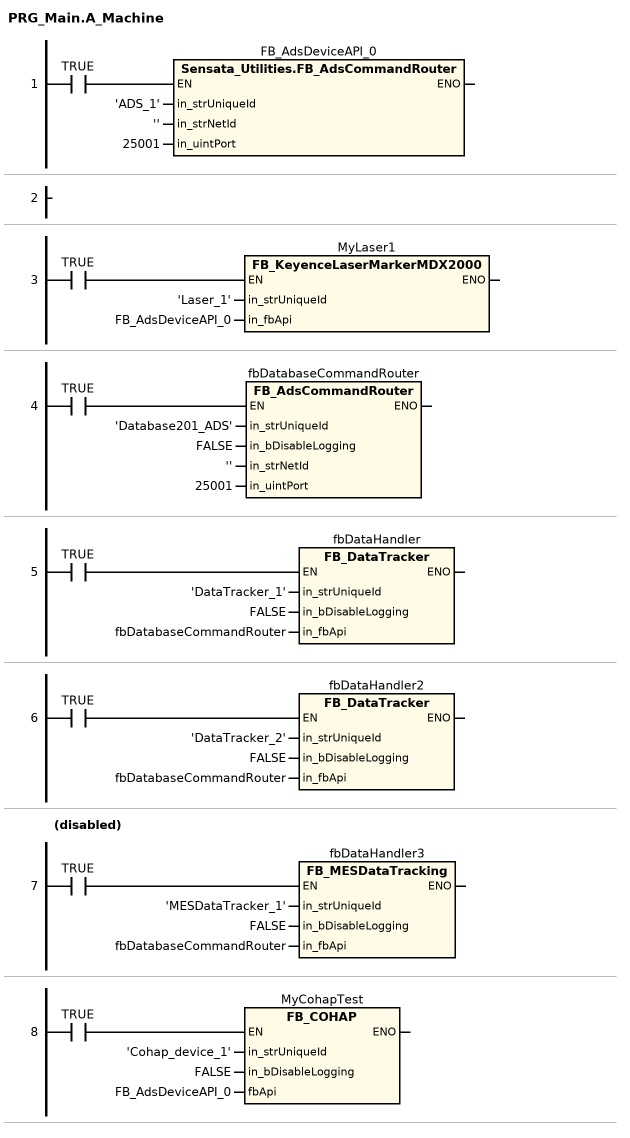
// NETWORK 1
FB_AdsDeviceAPI_0(in_strUniqueId := 'ADS_1', in_strNetId := '', in_uintPort := 25001); // Sensata_Utilities.FB_AdsCommandRouter

// NETWORK 2

// NETWORK 3
MyLaser1(in_strUniqueId := 'Laser_1', in_fbApi := FB_AdsDeviceAPI_0); // FB_KeyenceLaserMarkerMDX2000

// NETWORK 4
fbDatabaseCommandRouter(
    in_strUniqueId := 'Database201_ADS',
    in_bDisableLogging := FALSE,
    in_strNetId := '',
    in_uintPort := 25001); // FB_AdsCommandRouter

// NETWORK 5
fbDataHandler(
    in_strUniqueId := 'DataTracker_1',
    in_bDisableLogging := FALSE,
    in_fbApi := fbDatabaseCommandRouter); // FB_DataTracker

// NETWORK 6
fbDataHandler2(
    in_strUniqueId := 'DataTracker_2',
    in_bDisableLogging := FALSE,
    in_fbApi := fbDatabaseCommandRouter); // FB_DataTracker

// NETWORK 7 (disabled)
// fbDataHandler3(
//     in_strUniqueId := 'MESDataTracker_1',
//     in_bDisableLogging := FALSE,
//     in_fbApi := fbDatabaseCommandRouter); // FB_MESDataTracking

// NETWORK 8
MyCohapTest(in_strUniqueId := 'Cohap_device_1', in_bDisableLogging := FALSE, fbApi := FB_AdsDeviceAPI_0); // FB_COHAP
END_ACTION

ACTION A_Station1:
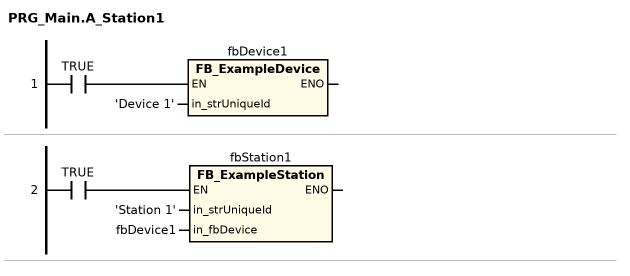
// NETWORK 1
fbDevice1(in_strUniqueId := 'Device 1'); // FB_ExampleDevice

// NETWORK 2
fbStation1(in_strUniqueId := 'Station 1', in_fbDevice := fbDevice1); // FB_ExampleStation
END_ACTION

ACTION A_Station2:
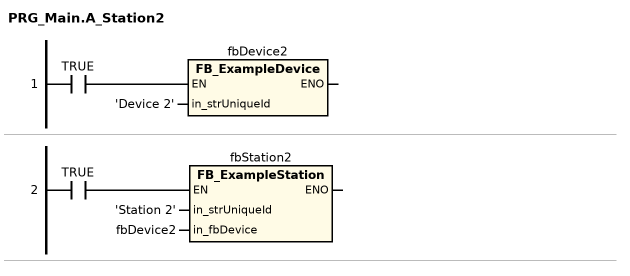
// NETWORK 1
fbDevice2(in_strUniqueId := 'Device 2'); // FB_ExampleDevice

// NETWORK 2
fbStation2(in_strUniqueId := 'Station 2', in_fbDevice := fbDevice2); // FB_ExampleStation
END_ACTION

ACTION A_Station3:
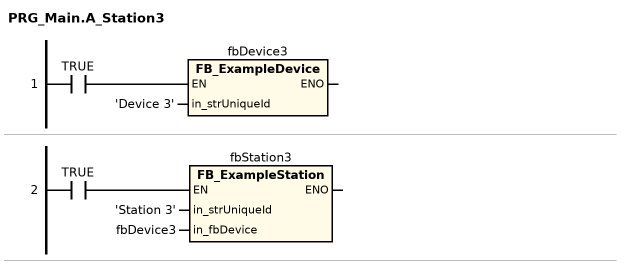
// NETWORK 1
fbDevice3(in_strUniqueId := 'Device 3'); // FB_ExampleDevice

// NETWORK 2
fbStation3(in_strUniqueId := 'Station 3', in_fbDevice := fbDevice3); // FB_ExampleStation
END_ACTION

ACTION A_Station4:
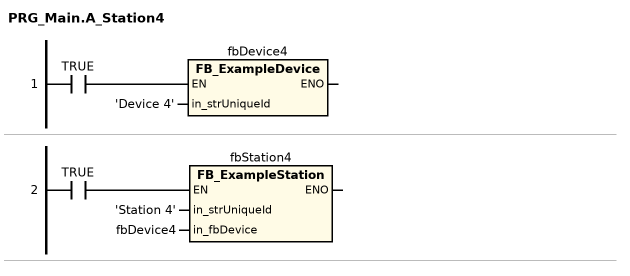
// NETWORK 1
fbDevice4(in_strUniqueId := 'Device 4'); // FB_ExampleDevice

// NETWORK 2
fbStation4(in_strUniqueId := 'Station 4', in_fbDevice := fbDevice4); // FB_ExampleStation
END_ACTION

END_PROGRAM

(* stored: Version 1.1.0.1, ProductVersion 3.1.4024.12
   POU PRG_Main: Id {b13f0be3-4c97-4edc-94e2-8c6f67cb8665}, SpecialFunc None
   Action A_CohapLDTesting: Id {d58812c4-a86f-4275-878d-6c8b63a41c0d}
   Action A_CohapLibraryTesting: Id {044fe8a4-3d4c-42ac-b64b-984c35c6fb2a}
   Action A_InitCohapMethodParams: Id {338b2860-1dc4-47ff-9b38-e01ddb531ef1}
   Action A_LaserMarkingParams: Id {23cacb87-0a2e-4564-9710-85ba7dafd933}
   Action A_Machine: Id {f2ef6f5c-8a40-4c62-8311-b3186050d362}
   Action A_Station1: Id {504119fa-b0a8-489a-9a37-499472501127}
   Action A_Station2: Id {21ea2e05-12d0-4cac-a384-2d35f55a53ab}
   Action A_Station3: Id {a8c1dd1b-134a-4dcf-b99f-4a08bcf13697}
   Action A_Station4: Id {f4929fa8-ed63-4a91-b73a-b4250062275b} *)
